{attribute 'qualified_only'}
{attribute 'strict'}
{attribute 'to_string'}
TYPE E_MOVER_SELECTOR :
(
	SELECT_MOVER_INDEX,
  SELECT_MOVER_AXIS_ID
);
END_TYPE

(* stored: Version 1.1.0.1
   DUT E_MOVER_SELECTOR: Id {b7bf8f43-092b-4f92-95d8-5d6eb0456619} *)
